TYPE U_AXIS_NC_PARAMETER_WRT :
UNION

  stCtrl              : ARRAY[1..MAX_AXIS] OF ST_NC_PARAMETER;

{IF defined (AXIS_MAP)}
  {info 'U_AXIS_NC_PARAMETER_WRT mapping activated'}
  byCtrl    AT %I*    : ARRAY[1..MAX_AXIS] OF
                        ARRAY[1..SIZEOF(ST_NC_PARAMETER)] OF BYTE;
{ELSE}
  byCtrl              : ARRAY[1..MAX_AXIS] OF
                        ARRAY[1..SIZEOF(ST_NC_PARAMETER)] OF BYTE;
{END_IF}
END_UNION
END_TYPE

(* stored: Version 1.1.0.1, ProductVersion 3.1.4024.15
   DUT U_AXIS_NC_PARAMETER_WRT: Id {0383247a-ba81-0347-342d-6eade186b955} *)
